TYPE ST_OperationPanel :
STRUCT
	bStart 						: BOOL;
	bEnable 					: BOOL;
	bDisable 					: BOOL;
	bReset 						: BOOL;
	bStop						: BOOL;
END_STRUCT
END_TYPE

(* stored: Version 1.1.0.1, ProductVersion 3.1.4024.12
   DUT ST_OperationPanel: Id {63276b87-f635-46fd-b38e-028b77e30390} *)
